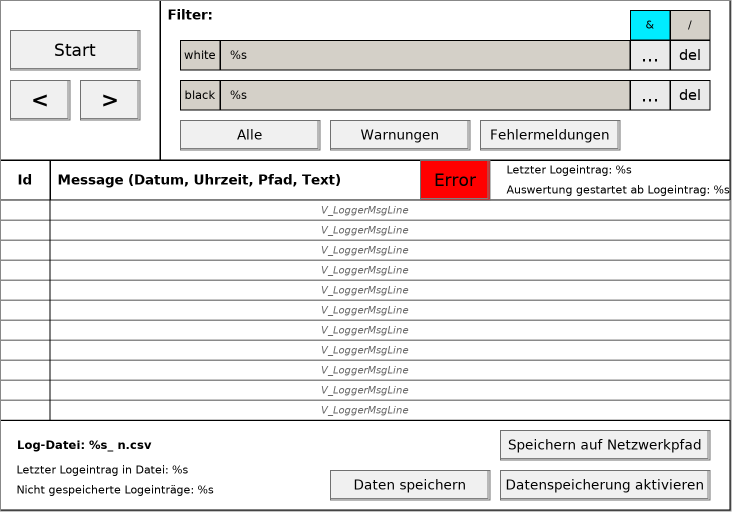
VISUALIZATION V_LoggerModul  // 732x512
VAR_IN_OUT
  fbLogger : FB_Logger;
END_VAR
    Rectangle (160,0 570x160)
    Rectangle (220,40 410x30), "%s", tooltip "'whitelist: Begriff1[;Begriff2[;Begriff3]]'", text variable: fbLogger.szVisuFilterWhite, colour toggle: fbLogger.bVisuFilterWhiteEnable
        OnMouseClick: execute { fbLogger.bVisuFilterWhiteEnable := TRUE; }
        OnMouseClick: write the text variable via Default
    Button (180,120 140x30), "Alle", colour toggle: fbLogger.iVisuFilterMsgTypInput <= 0
        OnMouseDown: execute { fbLogger.iVisuFilterMsgTypInput := 0; }
    Rectangle (670,40 40x30), "del", tooltip "löschen"
        OnMouseClick: execute { fbLogger.szVisuFilterWhite := ''; }
    Button (330,120 140x30), "Warnungen", colour toggle: fbLogger.iVisuFilterMsgTypInput = 1
        OnMouseDown: execute { fbLogger.iVisuFilterMsgTypInput := 1; }
    Button (480,120 140x30), "Fehlermeldungen", colour toggle: fbLogger.iVisuFilterMsgTypInput = 2
        OnMouseDown: execute { fbLogger.iVisuFilterMsgTypInput := 2; }
    Rectangle (220,80 410x30), "%s", tooltip "'black list: Begriff1[;Begriff2[;Begriff3]]'", text variable: fbLogger.szVisuFilterBlack, colour toggle: fbLogger.bVisuFilterBlackEnable
        OnMouseClick: execute { fbLogger.bVisuFilterBlackEnable := TRUE; }
        OnMouseClick: write the text variable via Default
    Rectangle (670,80 40x30), "del", tooltip "löschen"
        OnMouseClick: execute { fbLogger.szVisuFilterBlack := ''; }
    Rectangle (630,40 40x30), "...", tooltip "speichern/laden"
        OnMouseClick: execute { fbLogger.bVisuFilterWhiteEnable := TRUE; }
        OnMouseClick: change screen: V_LoggerFilterWhite
    Rectangle (630,80 40x30), "...", tooltip "speichern/laden"
        OnMouseClick: execute { fbLogger.bVisuFilterBlackEnable := TRUE; }
        OnMouseClick: change screen: V_LoggerFilterBlack
    Rectangle (0,0 160x160)
    Button (10,80 60x40), "<", invisible if: fbLogger.bVisuPrevPageInVisible
        toggle fbLogger.bVisuPrevPage
    Button (80,80 60x40), ">", invisible if: fbLogger.bVisuNextPageInVisible
        toggle fbLogger.bVisuNextPage
    Button (10,30 130x40), "Start", colour toggle: fbLogger.bVisuStart
        toggle fbLogger.bVisuStart
    Rectangle (0,160 50x40), "Id"
    Rectangle (50,160 680x40), "Message (Datum, Uhrzeit, Pfad, Text)"
    Frame (0,200 730x20)
        shows V_LoggerMsgLine(IOstLogMsg := fbLogger.astVisuLogMsg[1], IOiLogIdAct := fbLogger.nviLogId)
    Frame (0,220 730x20)
        shows V_LoggerMsgLine(IOstLogMsg := fbLogger.astVisuLogMsg[2], IOiLogIdAct := fbLogger.nviLogId)
    Frame (0,240 730x20)
        shows V_LoggerMsgLine(IOstLogMsg := fbLogger.astVisuLogMsg[3], IOiLogIdAct := fbLogger.nviLogId)
    Frame (0,260 730x20)
        shows V_LoggerMsgLine(IOstLogMsg := fbLogger.astVisuLogMsg[4], IOiLogIdAct := fbLogger.nviLogId)
    Frame (0,280 730x20)
        shows V_LoggerMsgLine(IOstLogMsg := fbLogger.astVisuLogMsg[5], IOiLogIdAct := fbLogger.nviLogId)
    Frame (0,300 730x20)
        shows V_LoggerMsgLine(IOstLogMsg := fbLogger.astVisuLogMsg[6], IOiLogIdAct := fbLogger.nviLogId)
    Frame (0,320 730x20)
        shows V_LoggerMsgLine(IOstLogMsg := fbLogger.astVisuLogMsg[7], IOiLogIdAct := fbLogger.nviLogId)
    Frame (0,340 730x20)
        shows V_LoggerMsgLine(IOstLogMsg := fbLogger.astVisuLogMsg[8], IOiLogIdAct := fbLogger.nviLogId)
    Frame (0,360 730x20)
        shows V_LoggerMsgLine(IOstLogMsg := fbLogger.astVisuLogMsg[9], IOiLogIdAct := fbLogger.nviLogId)
    Frame (0,380 730x20)
        shows V_LoggerMsgLine(IOstLogMsg := fbLogger.astVisuLogMsg[10], IOiLogIdAct := fbLogger.nviLogId)
    Rectangle (500,160 230x20), "Letzter Logeintrag: %s", text variable: fbLogger.nviLogId
    Rectangle (500,180 230x20), "Auswertung gestartet ab Logeintrag: %s", text variable: fbLogger.iVisuLogIdStart
    Rectangle (160,0 120x30), "Filter:"
    Button (420,160 70x40), "Error", invisible if: fbLogger.bVisuError = 0
    Frame (0,400 730x20)
        shows V_LoggerMsgLine(IOstLogMsg := fbLogger.astVisuLogMsg[11], IOiLogIdAct := fbLogger.nviLogId)
    Line (50,420) (50,200)
    Rectangle (180,40 40x30), "white", colour toggle: fbLogger.bVisuFilterWhiteEnable
        OnMouseClick: execute { fbLogger.bVisuFilterWhiteEnable := NOT fbLogger.bVisuFilterWhiteEnable; fbLogger.bVisuStart := TRUE; }
    Rectangle (670,10 40x30), "/", colour toggle: fbLogger.bVisuFilterWhiteMode_OR
        OnMouseClick: execute {
            fbLogger.bVisuFilterWhiteMode_OR := TRUE;
            fbLogger.bVisuFilterWhiteEnable := TRUE;
            fbLogger.bVisuStart := TRUE;
        }
    Rectangle (630,10 40x30), "&", colour toggle: fbLogger.bVisuFilterWhiteMode_OR
        OnMouseClick: execute {
            fbLogger.bVisuFilterWhiteMode_OR := FALSE;
            fbLogger.bVisuFilterWhiteEnable := TRUE;
            fbLogger.bVisuStart := TRUE;
        }
    Rectangle (180,80 40x30), "black", colour toggle: fbLogger.bVisuFilterBlackEnable
        OnMouseClick: execute { fbLogger.bVisuFilterBlackEnable := NOT fbLogger.bVisuFilterBlackEnable; fbLogger.bVisuStart := TRUE; }
    Rectangle (0,420 730x90)
    Rectangle (10,430 390x30), "Log-Datei: %s_ n.csv", text variable: fbLogger.fbFileWriteLogString.INszFileName, colour toggle: fbLogger.OUTbFileOpen
    Button (500,470 210x30), "Datenspeicherung aktivieren", tooltip "Daten werden automatisch gespeichert, wenn eine Mindestanzahl ungespeicherter Meldungen vorhanden ist.", colour toggle: fbLogger.nvbVisuFileWritingEnable
        toggle fbLogger.nvbVisuFileWritingEnable
    Button (330,470 160x30), "Daten speichern", tooltip "Daten sofort speichern", colour toggle: fbLogger.bVisuWriteToFileStart, invisible if: fbLogger.nvbVisuFileWritingEnable = 0
        OnMouseClick: execute { fbLogger.bVisuWriteToFileStart := TRUE; }
    Rectangle (10,460 230x20), "Letzter Logeintrag in Datei: %s", text variable: fbLogger.nviLogIdFileWriter
    Rectangle (10,480 220x20), "Nicht gespeicherte Logeinträge: %s", text variable: fbLogger.iFileWriterNumOfMsgsOpen, invisible if: fbLogger.nvbVisuFileWritingEnable = 0
    Button (500,430 210x30), "Speichern auf Netzwerkpfad", tooltip "Daten werden automatisch gespeichert, wenn eine Mindestanzahl ungespeicherter Meldungen vorhanden ist.", colour toggle: fbLogger.bVisuInitPathNetwork
        toggle fbLogger.bVisuInitPathNetwork
END_VISUALIZATION

(* stored: Version 1.1.0.1, ProductVersion 3.1.4018.10
   Visu V_LoggerModul: Id {4c56cb3e-bde1-4b74-a63f-ee1416a3d7de} *)
